Staubli VAL3: CloseAllFile.pgx

public program CloseAllFile()
begin

  call CloseFile(0)
  call CloseFile(1)
  call CloseFile(2)
  call CloseFile(3)
  call CloseFile(4)
  call CloseFile(5)
  call CloseFile(6)
  call CloseFile(7)
  call CloseFile(8)
  call CloseFile(9)
  delay(0)

end
